INTERFACE I_XtsIoEnvVar

METHOD GetCaGroupInterface : I_Mc2CaGroup
VAR_INPUT
	CAGroupNumber : INT;
END_VAR
END_METHOD

METHOD GetXPUInterface : I_TcIoXtsProcessingUnit
VAR_INPUT
	MyXts : INT;
END_VAR
END_METHOD

PROPERTY Initialised : BOOL
GET
END_GET
END_PROPERTY

END_INTERFACE

(* stored: Version 1.1.0.1
   Itf I_XtsIoEnvVar: Id {30a06d50-ef59-4bfa-9dd3-f949d401bfcc}
   Folder Commands: Id {1b5e6e83-f497-41ee-a2d2-91152888ebf2}
   Folder Status: Id {e000e9df-d48c-426c-8c4b-b82c6c436d9c}
   Method GetCaGroupInterface: Id {e5766ff7-d74d-4918-8c8c-b6404824695c}
   Method GetXPUInterface: Id {01d39393-68d5-4f22-a8cb-82a779c4b78e}
   Property Initialised: Id {6f24d56d-3c12-4d12-857a-612624baf1f9}
   Get Get: Id {bb6bc13b-7f6d-4c67-9fb0-330755e668e2} *)
